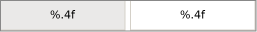
VISUALIZATION VISU_ConfigREAL4Entry  // 257x32
VAR_IN_OUT
    active : REAL;
    editable : REAL;
END_VAR
    Textfield (0,0 125x30), "%.4f", text variable: active, input disabled if: TRUE
    Textfield (130,0 125x30), "%.4f", text variable: editable, colour toggle: editable <> active
        OnMouseClick: write the text variable via Default
END_VISUALIZATION

(* stored: Version 1.1.0.1, ProductVersion 3.1.4018.5
   Visu VISU_ConfigREAL4Entry: Id {c9391b89-751e-4058-957f-24163f764b0d} *)
